{attribute 'OPC.UA.DA' := '1'}
{attribute 'OPC.UA.DA.StructuredType' := '1'}
{attribute 'pack_mode' := '1'} 
{attribute 'OPC.UA.AdditionalStructuredType.NamespaceName' := 'http://audi.com/OpcUa/CentralIm/'}
{attribute 'OPC.UA.AdditionalStructuredType.Id' := 'i=3010'}
TYPE ST_TargetValueType : UINT; END_TYPE

(* stored: Version 1.1.0.1, ProductVersion 3.1.4024.3
   DUT ST_TargetValueType: Id {cdd89684-23f5-4d8b-abe2-372268b347ba} *)
